// TIA Portal V18 export
// export: Created 2026-01-09T11:23:42.2246917Z, ExportSetting WithDefaults, DisplayName Totally Integrated Automation Portal, DisplayVersion V18 Update 5, DisplayName TIA Portal Openness, DisplayVersion V18 Update 5, DisplayName TIA Portal Teamcenter Gateway, DisplayVersion V18, DisplayName TIA Portal Version Control Interface, DisplayVersion V18, DisplayName SINAMICS Startdrive Advanced, DisplayVersion V18 SP2 Update 1, DisplayName SINAMICS Startdrive G110M, G120, G120C, G120D, G120P, G115D, DisplayVersion V18 SP2 Update 1, DisplayName SINAMICS Startdrive G130, G150, S120, S150, SINAMICS MV, S210, G220, S200, DisplayVersion V18 SP2 Update 1, DisplayName STEP 7 Professional, DisplayVersion V18 Update 5, DisplayName STEP 7 Safety, DisplayVersion V18, DisplayName WinCC Professional, DisplayVersion V18 Update 5
Screen "636 Analog Output"  1280x800, Number=636, Template=06Diagnosis
  ScreenLayer 
    TextField "文本域_2" at 88,182 size 115x32  StyleItem=TxtRight22, Text="PQW XXX"
    IOField "I/O 域_1" at 217,172 size 122x55  DataFormat=Decimal, FormatPattern=99999999, Mode=Output, StyleItem=I/O Display22
    IOField "I/O 域_2" at 355,172 size 122x55  DataFormat=Decimal, FormatPattern=99999999, Mode=Output, StyleItem=I/O Display22
    Button "按钮_1" at 896,725 size 128x75  Mode=Text, StyleItem=BtnActive20, TextOff="模拟量 输出信号 / AO Output Signal / Výstup AO Signál"
      on Click: ActivateScreen(Screen name := 616DP_Diagnosis, Object number := 0); SetTag(Tag := Sys_VersionManagement_HMIPageID, Value := 660)
